Staubli VAL3: place.pgx

program place(num x_nX, num x_nY, tool tGreifer)
begin
  // x,y [mm]


  pPlace.trsf.x = x_nX
  pPlace.trsf.y = x_nY



  movej(appro(pPlace,trApro),tGreifer, mUsedSpeed)
  movel(pPlace, tGreifer, mUsedSpeed)
  open(tGreifer)
  movel(appro(pPlace, trApro), tGreifer, mUsedSpeed)
  //logMsg("Objekt abgelegt")





end
